{attribute 'GeneratedUsingTerminal: EL6201-0000-0017'}
{attribute addProperty BoxType "EL6201-0000-0017"}
{attribute addProperty Id "Slave_18A_DO0BOOL1Slave_18A_DO1BOOL1Slave_18A_DO2BOOL1Slave_18A_DO3BOOL1Slave_18B_DO0BOOL1Slave_18B_DO1BOOL1Slave_18B_DO2BOOL1Slave_18B_DO3BOOL1"}
{attribute addProperty CRC "2315049256"}
{attribute addProperty Size "8"}
TYPE Slave_18_Outputs_89FCD928 :
STRUCT
	{attribute addProperty Name "Slave_18A_DO0"}
	Slave_18A_DO0 : BOOL;
	{attribute addProperty Name "Slave_18A_DO1"}
	Slave_18A_DO1 : BOOL;
	{attribute addProperty Name "Slave_18A_DO2"}
	Slave_18A_DO2 : BOOL;
	{attribute addProperty Name "Slave_18A_DO3"}
	Slave_18A_DO3 : BOOL;
	{attribute addProperty Name "Slave_18B_DO0"}
	Slave_18B_DO0 : BOOL;
	{attribute addProperty Name "Slave_18B_DO1"}
	Slave_18B_DO1 : BOOL;
	{attribute addProperty Name "Slave_18B_DO2"}
	Slave_18B_DO2 : BOOL;
	{attribute addProperty Name "Slave_18B_DO3"}
	Slave_18B_DO3 : BOOL;
END_STRUCT
END_TYPE

(* stored: Version 1.2.0.0, ProductVersion 3.1.4024.9
   DUT Slave_18_Outputs_89FCD928: Id {f0a37465-28d5-4012-a287-04691109f109} *)
